% RSLogix 500 project JBT BIN SETTON ORIGINAL - COPY_BAK001.RSS, saved by version 10.00.00.00 %
PROJECT "JBT BIN"    % processor: MicroLogix 1200 %

PROGRAM FILES
  LAD 2   10 rungs
  LAD 3   7 rungs
  LAD 4   11 rungs
  LAD 5   33 rungs
  LAD 6   26 rungs
  LAD 7   16 rungs
  LAD 8   14 rungs
  LAD 9   43 rungs
  LAD 10   16 rungs
  LAD 11   9 rungs

DATA FILES
  O0 OUTPUT  6 elements
  I1 INPUT  6 elements
  S2 STATUS  66 elements
  B3 BINARY  5 elements
  T4 TIMER  35 elements
  C5 COUNTER  1 elements
  R6 CONTROL  1 elements
  N7 INTEGER  34 elements
  F8 FLOAT  1 elements
  L9   1 elements
  L10   2 elements

LADDER 2
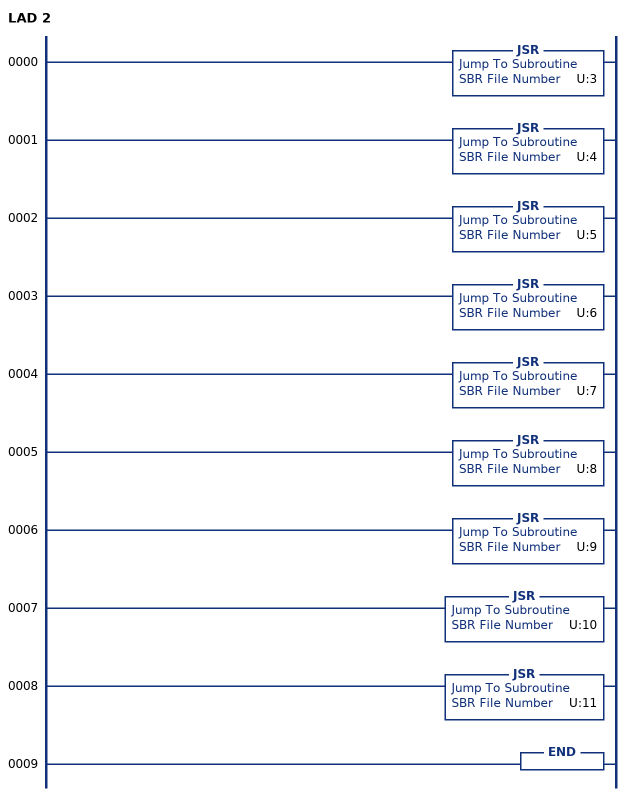
% Rung: 0 %
SOR JSR U:3 EOR
% Rung: 1 %
SOR JSR U:4 EOR
% Rung: 2 %
SOR JSR U:5 EOR
% Rung: 3 %
SOR JSR U:6 EOR
% Rung: 4 %
SOR JSR U:7 EOR
% Rung: 5 %
SOR JSR U:8 EOR
% Rung: 6 %
SOR JSR U:9 EOR
% Rung: 7 %
SOR JSR U:10 EOR
% Rung: 8 %
SOR JSR U:11 EOR
% Rung: 9 %
SOR END EOR

LADDER 3
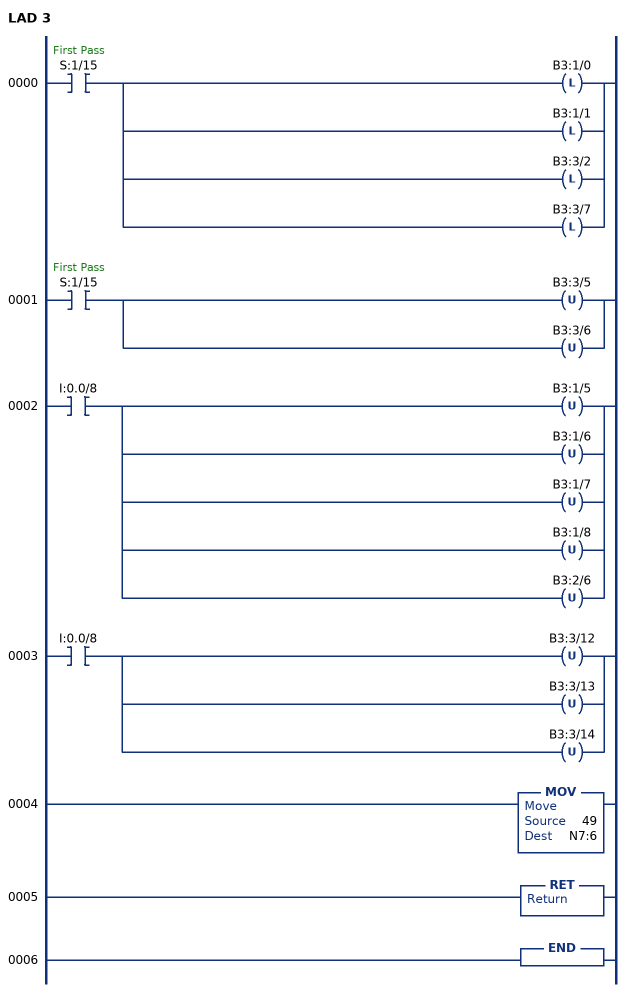
% Rung: 0 %
SOR XIC S:1/15 BST OTL B3:1/0 NXB BST OTL B3:1/1 NXB BST OTL B3:3/2 NXB OTL B3:3/7 BND BND BND EOR
%   S:1/15  "First Pass" %
% Rung: 1 %
SOR XIC S:1/15 BST OTU B3:3/5 NXB OTU B3:3/6 BND EOR
%   S:1/15  "First Pass" %
% Rung: 2 %
SOR XIC I:0.0/8 BST OTU B3:1/5 NXB BST OTU B3:1/6 NXB OTU B3:1/7 NXB BST OTU B3:1/8 NXB OTU B3:2/6 BND BND BND EOR
% Rung: 3 %
SOR XIC I:0.0/8 BST OTU B3:3/12 NXB OTU B3:3/13 NXB OTU B3:3/14 BND EOR
% Rung: 4 %
SOR MOV 49 N7:6 EOR
% Rung: 5 %
SOR RET EOR
% Rung: 6 %
SOR END EOR

LADDER 4
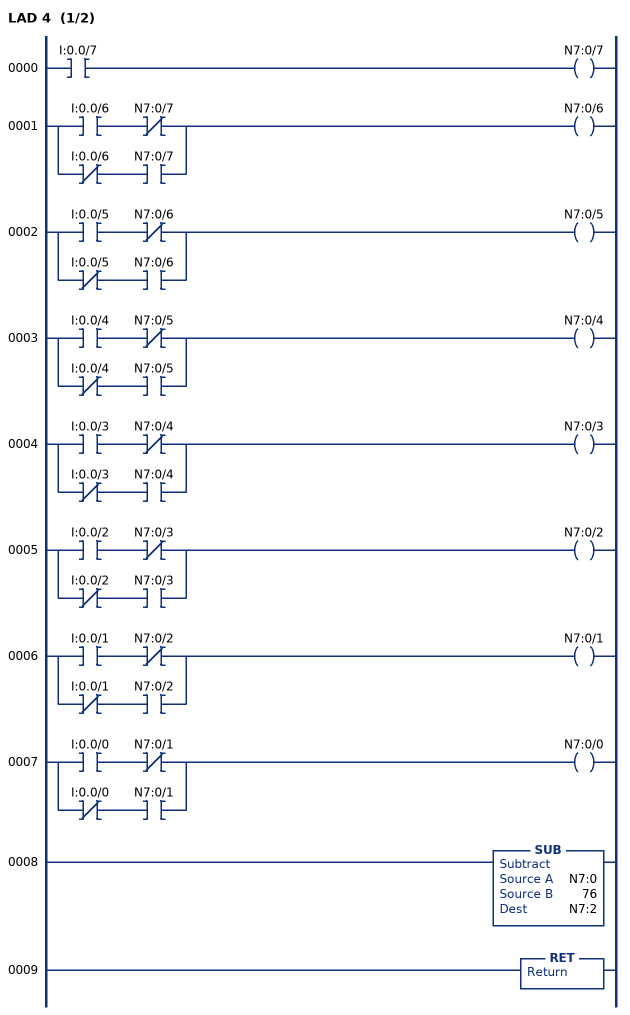
% Rung: 0 %
SOR XIC I:0.0/7 OTE N7:0/7 EOR
% Rung: 1 %
SOR BST XIC I:0.0/6 XIO N7:0/7 NXB XIO I:0.0/6 XIC N7:0/7 BND OTE N7:0/6 EOR
% Rung: 2 %
SOR BST XIC I:0.0/5 XIO N7:0/6 NXB XIO I:0.0/5 XIC N7:0/6 BND OTE N7:0/5 EOR
% Rung: 3 %
SOR BST XIC I:0.0/4 XIO N7:0/5 NXB XIO I:0.0/4 XIC N7:0/5 BND OTE N7:0/4 EOR
% Rung: 4 %
SOR BST XIC I:0.0/3 XIO N7:0/4 NXB XIO I:0.0/3 XIC N7:0/4 BND OTE N7:0/3 EOR
% Rung: 5 %
SOR BST XIC I:0.0/2 XIO N7:0/3 NXB XIO I:0.0/2 XIC N7:0/3 BND OTE N7:0/2 EOR
% Rung: 6 %
SOR BST XIC I:0.0/1 XIO N7:0/2 NXB XIO I:0.0/1 XIC N7:0/2 BND OTE N7:0/1 EOR
% Rung: 7 %
SOR BST XIC I:0.0/0 XIO N7:0/1 NXB XIO I:0.0/0 XIC N7:0/1 BND OTE N7:0/0 EOR
% Rung: 8 %
SOR SUB N7:0 76 N7:2 EOR
% Rung: 9 %
SOR RET EOR

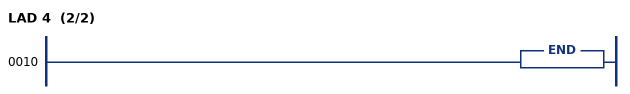
% Rung: 10 %
SOR END EOR

LADDER 5
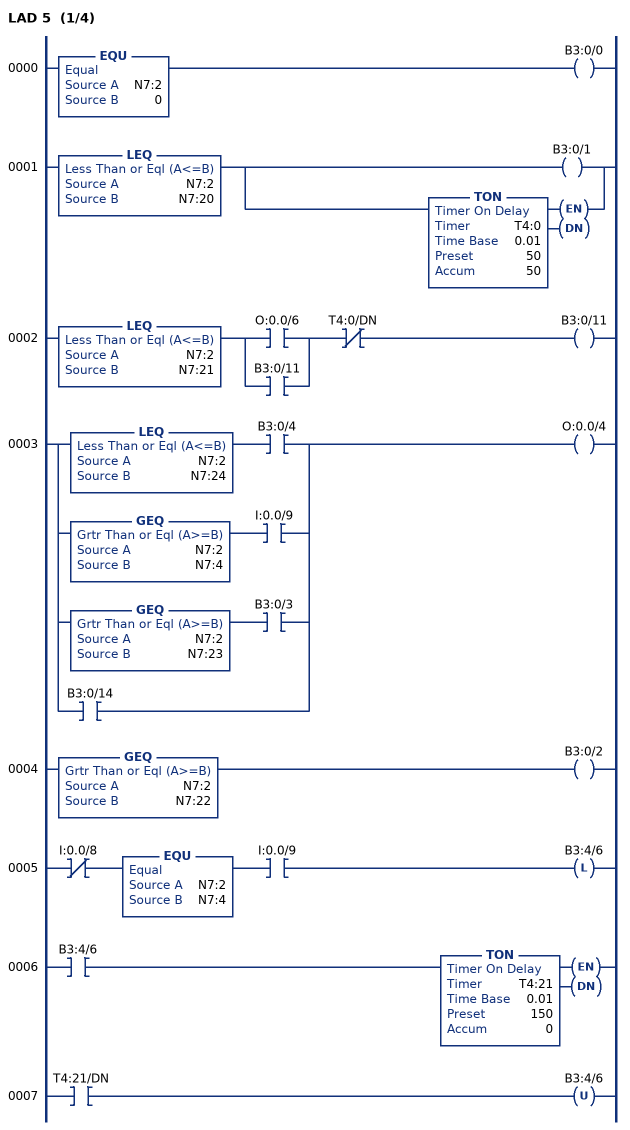
% Rung: 0 %
SOR EQU N7:2 0 OTE B3:0/0 EOR
% Rung: 1 %
SOR LEQ N7:2 N7:20 BST OTE B3:0/1 NXB TON T4:0 0.01 50 50 BND EOR
% Rung: 2 %
SOR LEQ N7:2 N7:21 BST XIC O:0.0/6 NXB XIC B3:0/11 BND XIO T4:0/DN OTE B3:0/11 EOR
% Rung: 3 %
SOR BST LEQ N7:2 N7:24 XIC B3:0/4 NXB GEQ N7:2 N7:4 XIC I:0.0/9 NXB BST GEQ N7:2 N7:23 XIC B3:0/3 NXB XIC B3:0/14 BND BND OTE O:0.0/4 EOR
% Rung: 4 %
SOR GEQ N7:2 N7:22 OTE B3:0/2 EOR
% Rung: 5 %
SOR XIO I:0.0/8 EQU N7:2 N7:4 XIC I:0.0/9 OTL B3:4/6 EOR
% Rung: 6 %
SOR XIC B3:4/6 TON T4:21 0.01 150 0 EOR
% Rung: 7 %
SOR XIC T4:21/DN OTU B3:4/6 EOR

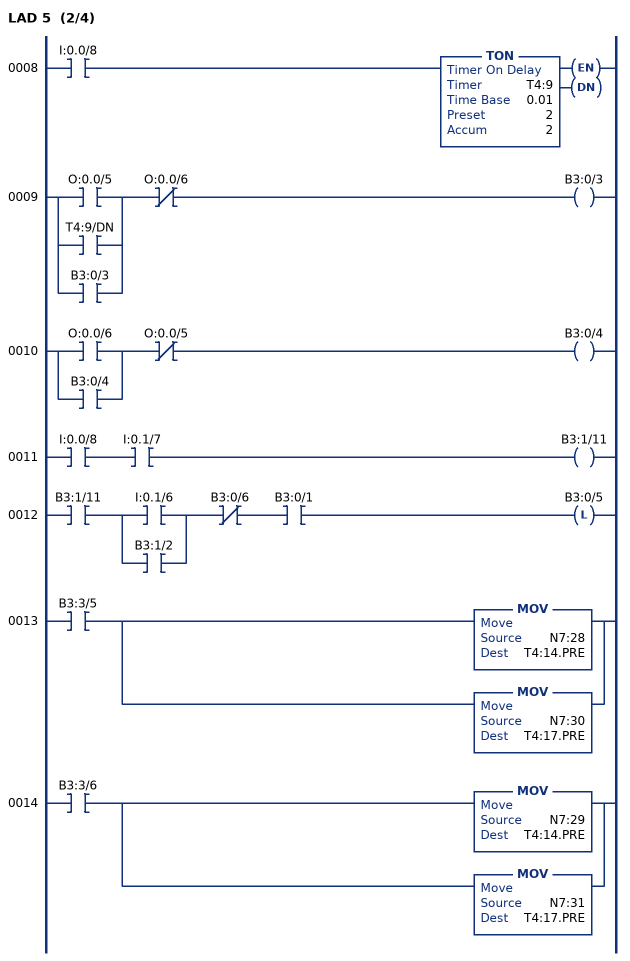
% Rung: 8 %
SOR XIC I:0.0/8 TON T4:9 0.01 2 2 EOR
% Rung: 9 %
SOR BST XIC O:0.0/5 NXB XIC T4:9/DN NXB XIC B3:0/3 BND XIO O:0.0/6 OTE B3:0/3 EOR
% Rung: 10 %
SOR BST XIC O:0.0/6 NXB XIC B3:0/4 BND XIO O:0.0/5 OTE B3:0/4 EOR
% Rung: 11 %
SOR XIC I:0.0/8 XIC I:0.1/7 OTE B3:1/11 EOR
% Rung: 12 %
SOR XIC B3:1/11 BST XIC I:0.1/6 NXB XIC B3:1/2 BND XIO B3:0/6 XIC B3:0/1 OTL B3:0/5 EOR
% Rung: 13 %
SOR XIC B3:3/5 BST MOV N7:28 T4:14.PRE NXB MOV N7:30 T4:17.PRE BND EOR
% Rung: 14 %
SOR XIC B3:3/6 BST MOV N7:29 T4:14.PRE NXB MOV N7:31 T4:17.PRE BND EOR

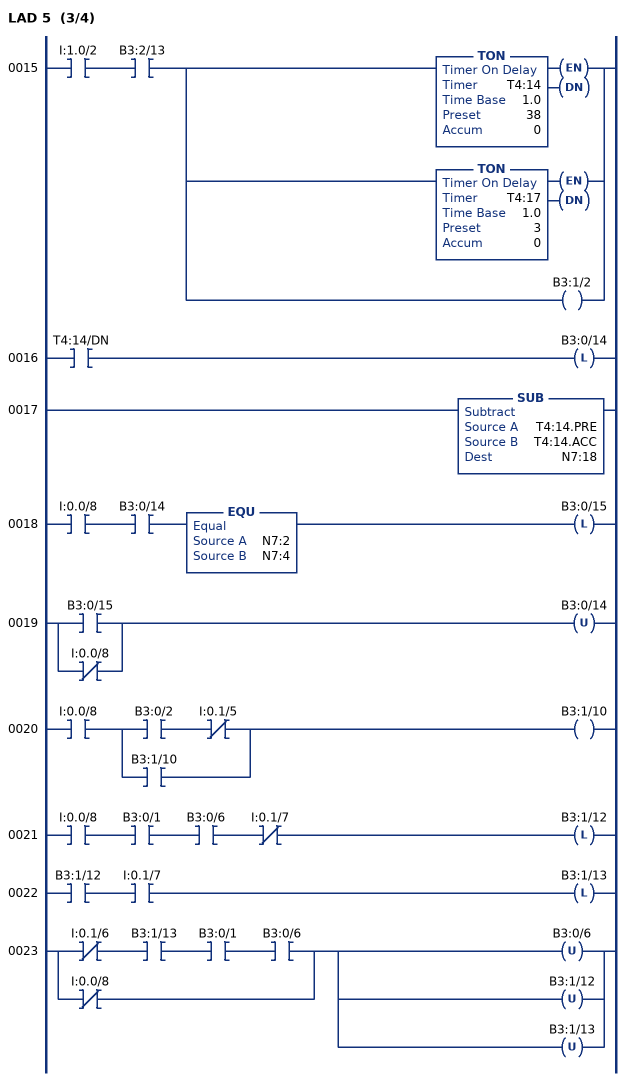
% Rung: 15 %
SOR XIC I:1.0/2 XIC B3:2/13 BST TON T4:14 1.0 38 0 NXB TON T4:17 1.0 3 0 NXB OTE B3:1/2 BND EOR
% Rung: 16 %
SOR XIC T4:14/DN OTL B3:0/14 EOR
% Rung: 17 %
SOR SUB T4:14.PRE T4:14.ACC N7:18 EOR
% Rung: 18 %
SOR XIC I:0.0/8 XIC B3:0/14 EQU N7:2 N7:4 OTL B3:0/15 EOR
% Rung: 19 %
SOR BST XIC B3:0/15 NXB XIO I:0.0/8 BND OTU B3:0/14 EOR
% Rung: 20 %
SOR XIC I:0.0/8 BST XIC B3:0/2 XIO I:0.1/5 NXB XIC B3:1/10 BND OTE B3:1/10 EOR
% Rung: 21 %
SOR XIC I:0.0/8 XIC B3:0/1 XIC B3:0/6 XIO I:0.1/7 OTL B3:1/12 EOR
% Rung: 22 %
SOR XIC B3:1/12 XIC I:0.1/7 OTL B3:1/13 EOR
% Rung: 23 %
SOR BST XIO I:0.1/6 XIC B3:1/13 XIC B3:0/1 XIC B3:0/6 NXB XIO I:0.0/8 BND BST OTU B3:0/6 NXB BST OTU B3:1/12 NXB OTU B3:1/13 BND BND EOR

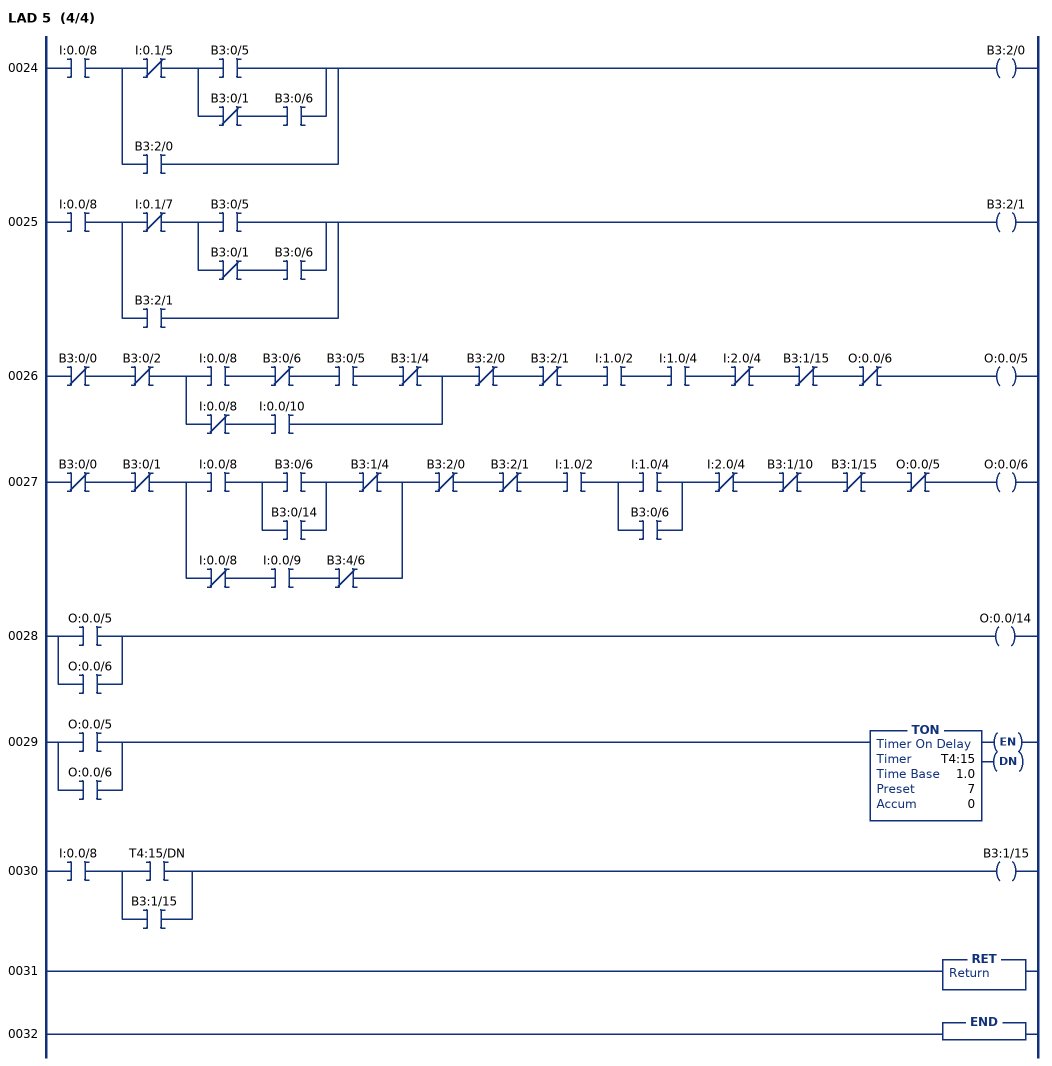
% Rung: 24 %
SOR XIC I:0.0/8 BST XIO I:0.1/5 BST XIC B3:0/5 NXB XIO B3:0/1 XIC B3:0/6 BND NXB XIC B3:2/0 BND OTE B3:2/0 EOR
% Rung: 25 %
SOR XIC I:0.0/8 BST XIO I:0.1/7 BST XIC B3:0/5 NXB XIO B3:0/1 XIC B3:0/6 BND NXB XIC B3:2/1 BND OTE B3:2/1 EOR
% Rung: 26 %
SOR XIO B3:0/0 XIO B3:0/2 BST XIC I:0.0/8 XIO B3:0/6 XIC B3:0/5 XIO B3:1/4 NXB XIO I:0.0/8 XIC I:0.0/10 BND XIO B3:2/0 XIO B3:2/1 XIC I:1.0/2 XIC I:1.0/4 XIO I:2.0/4 XIO B3:1/15 XIO O:0.0/6 OTE O:0.0/5 EOR
% Rung: 27 %
SOR XIO B3:0/0 XIO B3:0/1 BST XIC I:0.0/8 BST XIC B3:0/6 NXB XIC B3:0/14 BND XIO B3:1/4 NXB XIO I:0.0/8 XIC I:0.0/9 XIO B3:4/6 BND XIO B3:2/0 XIO B3:2/1 XIC I:1.0/2 BST XIC I:1.0/4 NXB XIC B3:0/6 BND XIO I:2.0/4 XIO B3:1/10 XIO B3:1/15 XIO O:0.0/5 OTE O:0.0/6 EOR
% Rung: 28 %
SOR BST XIC O:0.0/5 NXB XIC O:0.0/6 BND OTE O:0.0/14 EOR
% Rung: 29 %
SOR BST XIC O:0.0/5 NXB XIC O:0.0/6 BND TON T4:15 1.0 7 0 EOR
% Rung: 30 %
SOR XIC I:0.0/8 BST XIC T4:15/DN NXB XIC B3:1/15 BND OTE B3:1/15 EOR
% Rung: 31 %
SOR RET EOR
% Rung: 32 %
SOR END EOR

LADDER 6
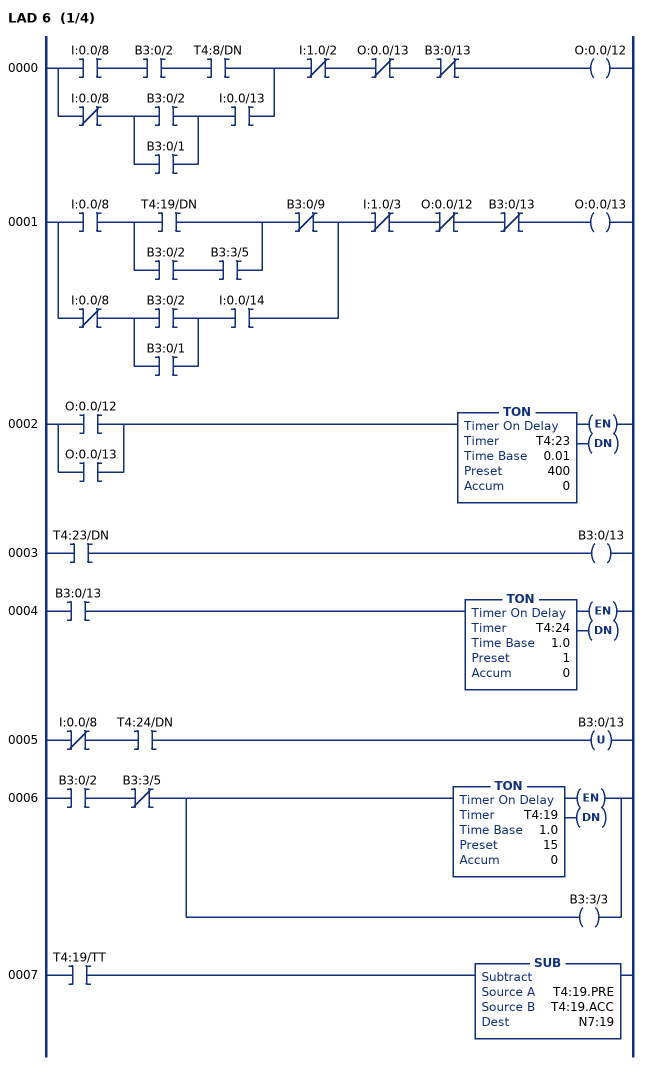
% Rung: 0 %
SOR BST XIC I:0.0/8 XIC B3:0/2 XIC T4:8/DN NXB XIO I:0.0/8 BST XIC B3:0/2 NXB XIC B3:0/1 BND XIC I:0.0/13 BND XIO I:1.0/2 XIO O:0.0/13 XIO B3:0/13 OTE O:0.0/12 EOR
% Rung: 1 %
SOR BST XIC I:0.0/8 BST XIC T4:19/DN NXB XIC B3:0/2 XIC B3:3/5 BND XIO B3:0/9 NXB XIO I:0.0/8 BST XIC B3:0/2 NXB XIC B3:0/1 BND XIC I:0.0/14 BND XIO I:1.0/3 XIO O:0.0/12 XIO B3:0/13 OTE O:0.0/13 EOR
% Rung: 2 %
SOR BST XIC O:0.0/12 NXB XIC O:0.0/13 BND TON T4:23 0.01 400 0 EOR
% Rung: 3 %
SOR XIC T4:23/DN OTE B3:0/13 EOR
% Rung: 4 %
SOR XIC B3:0/13 TON T4:24 1.0 1 0 EOR
% Rung: 5 %
SOR XIO I:0.0/8 XIC T4:24/DN OTU B3:0/13 EOR
% Rung: 6 %
SOR XIC B3:0/2 XIO B3:3/5 BST TON T4:19 1.0 15 0 NXB OTE B3:3/3 BND EOR
% Rung: 7 %
SOR XIC T4:19/TT SUB T4:19.PRE T4:19.ACC N7:19 EOR

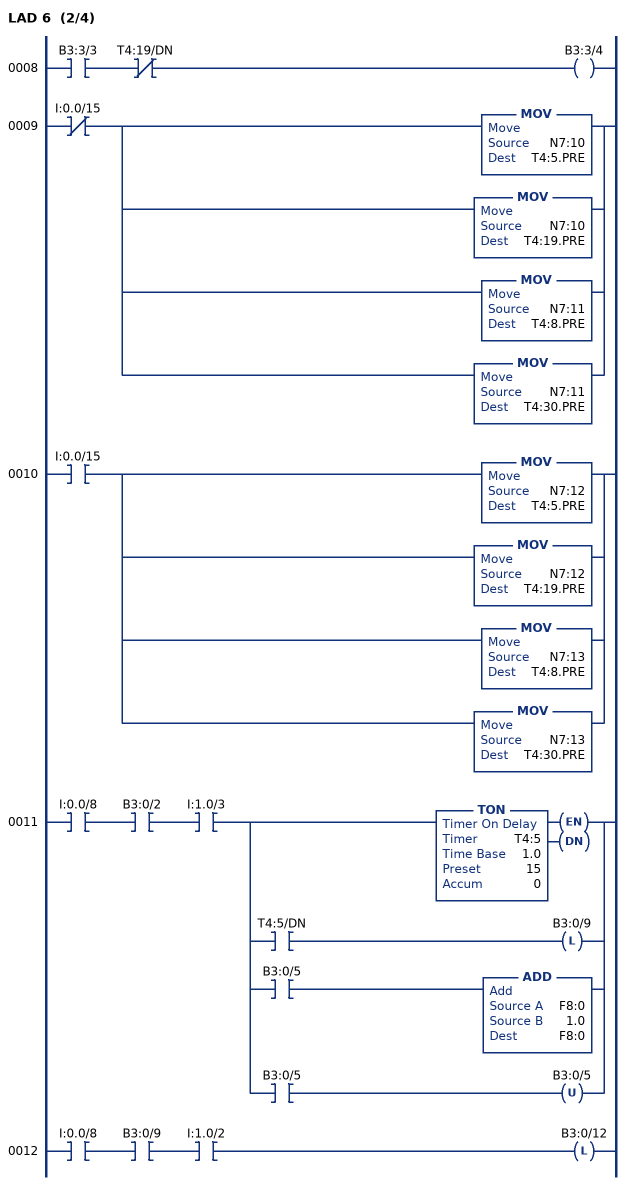
% Rung: 8 %
SOR XIC B3:3/3 XIO T4:19/DN OTE B3:3/4 EOR
% Rung: 9 %
SOR XIO I:0.0/15 BST MOV N7:10 T4:5.PRE NXB MOV N7:10 T4:19.PRE NXB MOV N7:11 T4:8.PRE NXB MOV N7:11 T4:30.PRE BND EOR
% Rung: 10 %
SOR XIC I:0.0/15 BST MOV N7:12 T4:5.PRE NXB MOV N7:12 T4:19.PRE NXB MOV N7:13 T4:8.PRE NXB MOV N7:13 T4:30.PRE BND EOR
% Rung: 11 %
SOR XIC I:0.0/8 XIC B3:0/2 XIC I:1.0/3 BST TON T4:5 1.0 15 0 NXB XIC T4:5/DN OTL B3:0/9 NXB BST XIC B3:0/5 ADD F8:0 1.0 F8:0 NXB XIC B3:0/5 OTU B3:0/5 BND BND EOR
% Rung: 12 %
SOR XIC I:0.0/8 XIC B3:0/9 XIC I:1.0/2 OTL B3:0/12 EOR

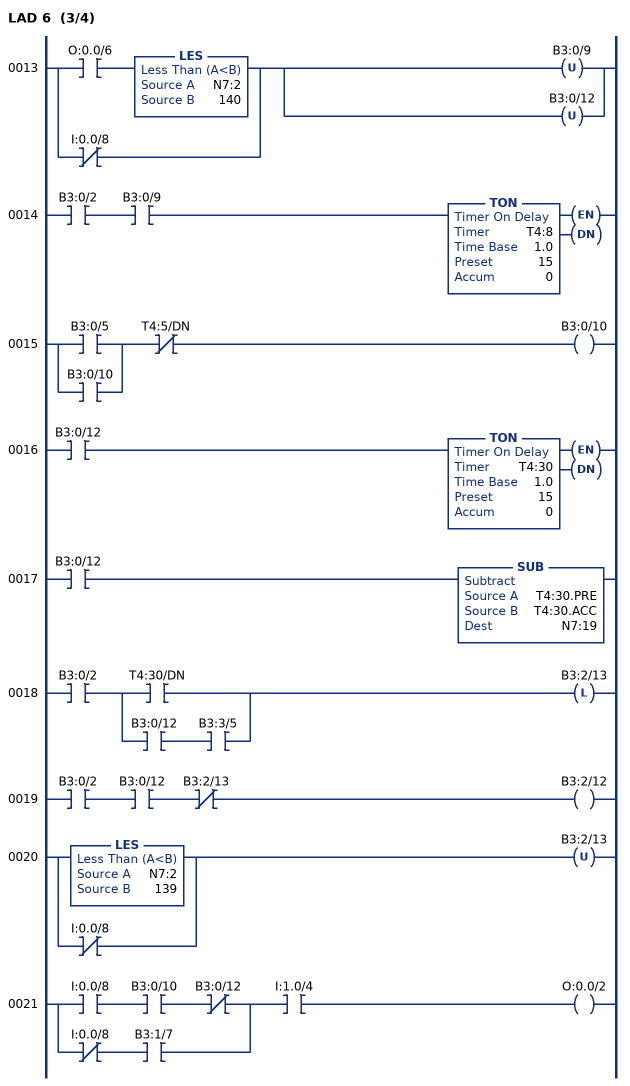
% Rung: 13 %
SOR BST XIC O:0.0/6 LES N7:2 140 NXB XIO I:0.0/8 BND BST OTU B3:0/9 NXB OTU B3:0/12 BND EOR
% Rung: 14 %
SOR XIC B3:0/2 XIC B3:0/9 TON T4:8 1.0 15 0 EOR
% Rung: 15 %
SOR BST XIC B3:0/5 NXB XIC B3:0/10 BND XIO T4:5/DN OTE B3:0/10 EOR
% Rung: 16 %
SOR XIC B3:0/12 TON T4:30 1.0 15 0 EOR
% Rung: 17 %
SOR XIC B3:0/12 SUB T4:30.PRE T4:30.ACC N7:19 EOR
% Rung: 18 %
SOR XIC B3:0/2 BST XIC T4:30/DN NXB XIC B3:0/12 XIC B3:3/5 BND OTL B3:2/13 EOR
% Rung: 19 %
SOR XIC B3:0/2 XIC B3:0/12 XIO B3:2/13 OTE B3:2/12 EOR
% Rung: 20 %
SOR BST LES N7:2 139 NXB XIO I:0.0/8 BND OTU B3:2/13 EOR
% Rung: 21 %
SOR BST XIC I:0.0/8 XIC B3:0/10 XIO B3:0/12 NXB XIO I:0.0/8 XIC B3:1/7 BND XIC I:1.0/4 OTE O:0.0/2 EOR

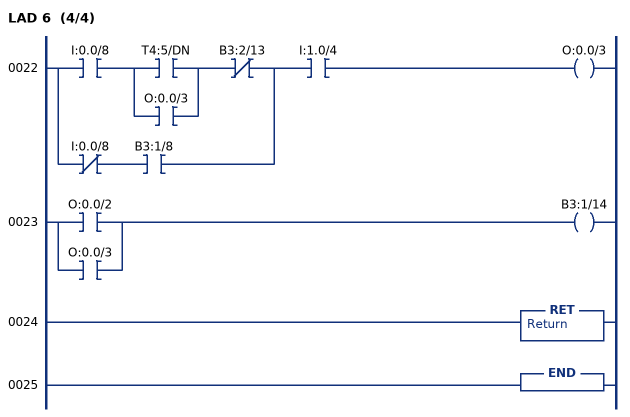
% Rung: 22 %
SOR BST XIC I:0.0/8 BST XIC T4:5/DN NXB XIC O:0.0/3 BND XIO B3:2/13 NXB XIO I:0.0/8 XIC B3:1/8 BND XIC I:1.0/4 OTE O:0.0/3 EOR
% Rung: 23 %
SOR BST XIC O:0.0/2 NXB XIC O:0.0/3 BND OTE B3:1/14 EOR
% Rung: 24 %
SOR RET EOR
% Rung: 25 %
SOR END EOR

LADDER 7
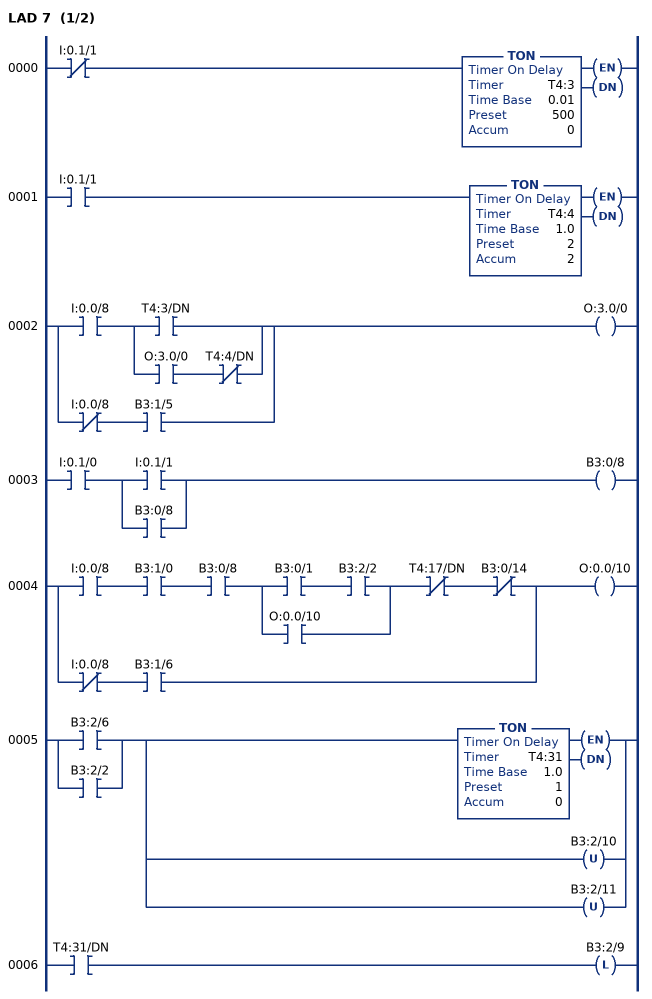
% Rung: 0 %
SOR XIO I:0.1/1 TON T4:3 0.01 500 0 EOR
% Rung: 1 %
SOR XIC I:0.1/1 TON T4:4 1.0 2 2 EOR
% Rung: 2 %
SOR BST XIC I:0.0/8 BST XIC T4:3/DN NXB XIC O:3.0/0 XIO T4:4/DN BND NXB XIO I:0.0/8 XIC B3:1/5 BND OTE O:3.0/0 EOR
% Rung: 3 %
SOR XIC I:0.1/0 BST XIC I:0.1/1 NXB XIC B3:0/8 BND OTE B3:0/8 EOR
% Rung: 4 %
SOR BST XIC I:0.0/8 XIC B3:1/0 XIC B3:0/8 BST XIC B3:0/1 XIC B3:2/2 NXB XIC O:0.0/10 BND XIO T4:17/DN XIO B3:0/14 NXB XIO I:0.0/8 XIC B3:1/6 BND OTE O:0.0/10 EOR
% Rung: 5 %
SOR BST XIC B3:2/6 NXB XIC B3:2/2 BND BST TON T4:31 1.0 1 0 NXB BST OTU B3:2/10 NXB OTU B3:2/11 BND BND EOR
% Rung: 6 %
SOR XIC T4:31/DN OTL B3:2/9 EOR

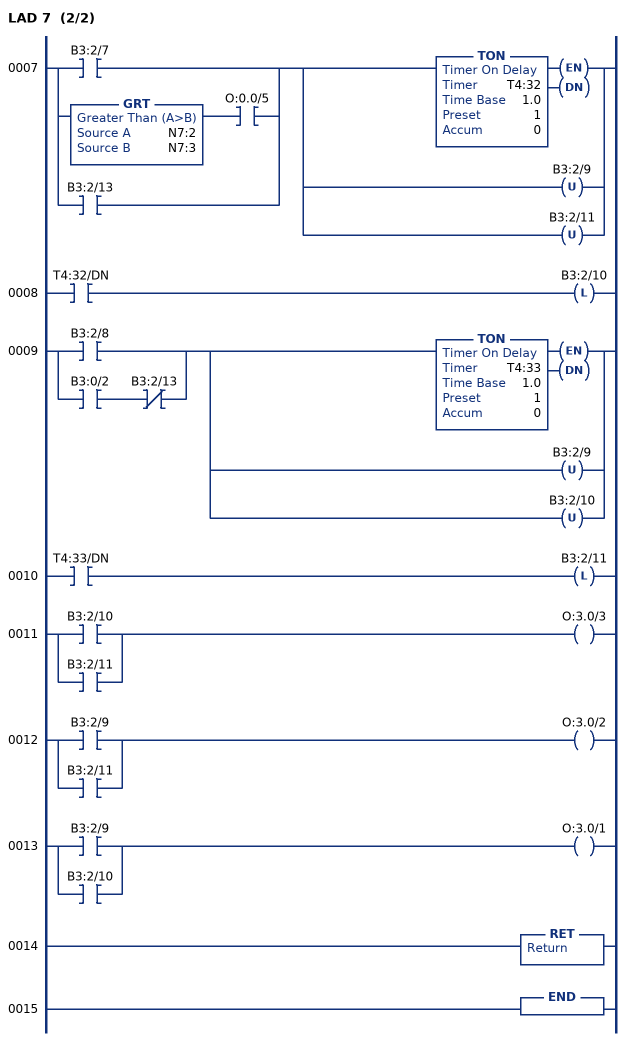
% Rung: 7 %
SOR BST BST XIC B3:2/7 NXB GRT N7:2 N7:3 XIC O:0.0/5 BND NXB XIC B3:2/13 BND BST TON T4:32 1.0 1 0 NXB BST OTU B3:2/9 NXB OTU B3:2/11 BND BND EOR
% Rung: 8 %
SOR XIC T4:32/DN OTL B3:2/10 EOR
% Rung: 9 %
SOR BST XIC B3:2/8 NXB XIC B3:0/2 XIO B3:2/13 BND BST TON T4:33 1.0 1 0 NXB BST OTU B3:2/9 NXB OTU B3:2/10 BND BND EOR
% Rung: 10 %
SOR XIC T4:33/DN OTL B3:2/11 EOR
% Rung: 11 %
SOR BST XIC B3:2/10 NXB XIC B3:2/11 BND OTE O:3.0/3 EOR
% Rung: 12 %
SOR BST XIC B3:2/9 NXB XIC B3:2/11 BND OTE O:3.0/2 EOR
% Rung: 13 %
SOR BST XIC B3:2/9 NXB XIC B3:2/10 BND OTE O:3.0/1 EOR
% Rung: 14 %
SOR RET EOR
% Rung: 15 %
SOR END EOR

LADDER 8
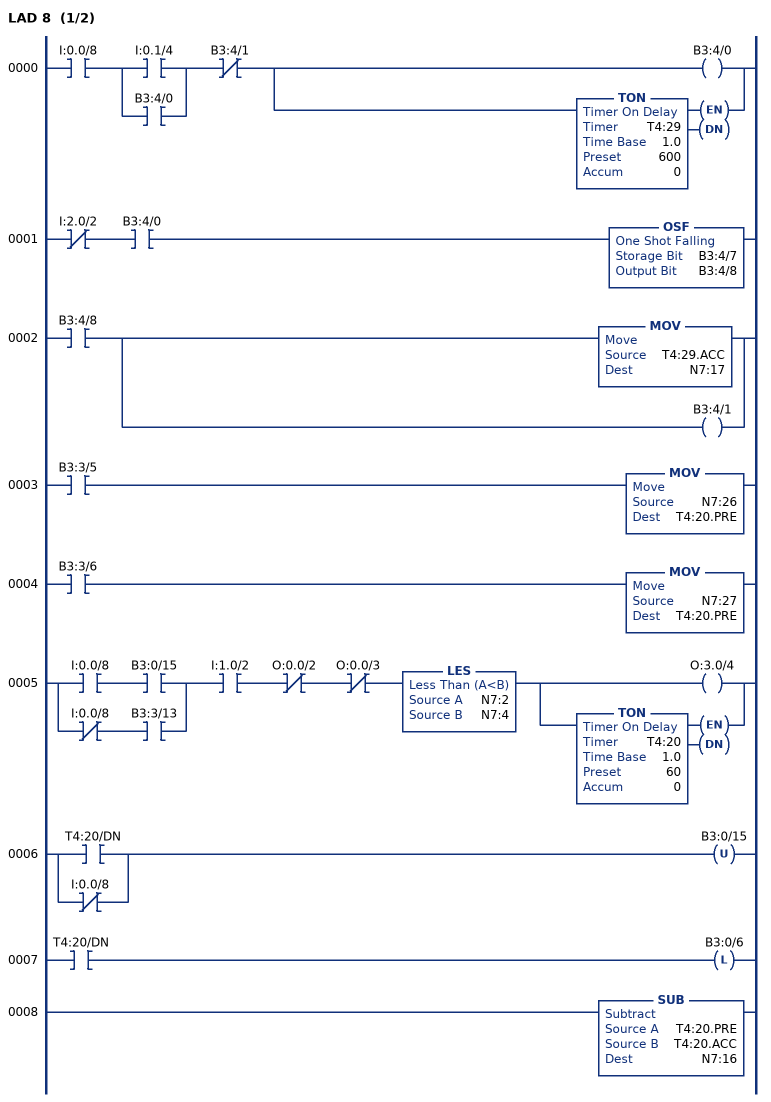
% Rung: 0 %
SOR XIC I:0.0/8 BST XIC I:0.1/4 NXB XIC B3:4/0 BND XIO B3:4/1 BST OTE B3:4/0 NXB TON T4:29 1.0 600 0 BND EOR
% Rung: 1 %
SOR XIO I:2.0/2 XIC B3:4/0 OSF B3:4/7 B3:4/8 EOR
% Rung: 2 %
SOR XIC B3:4/8 BST MOV T4:29.ACC N7:17 NXB OTE B3:4/1 BND EOR
% Rung: 3 %
SOR XIC B3:3/5 MOV N7:26 T4:20.PRE EOR
% Rung: 4 %
SOR XIC B3:3/6 MOV N7:27 T4:20.PRE EOR
% Rung: 5 %
SOR BST XIC I:0.0/8 XIC B3:0/15 NXB XIO I:0.0/8 XIC B3:3/13 BND XIC I:1.0/2 XIO O:0.0/2 XIO O:0.0/3 LES N7:2 N7:4 BST OTE O:3.0/4 NXB TON T4:20 1.0 60 0 BND EOR
% Rung: 6 %
SOR BST XIC T4:20/DN NXB XIO I:0.0/8 BND OTU B3:0/15 EOR
% Rung: 7 %
SOR XIC T4:20/DN OTL B3:0/6 EOR
% Rung: 8 %
SOR SUB T4:20.PRE T4:20.ACC N7:16 EOR

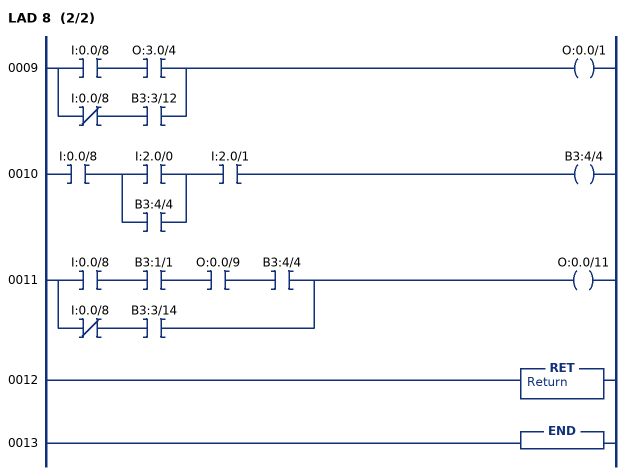
% Rung: 9 %
SOR BST XIC I:0.0/8 XIC O:3.0/4 NXB XIO I:0.0/8 XIC B3:3/12 BND OTE O:0.0/1 EOR
% Rung: 10 %
SOR XIC I:0.0/8 BST XIC I:2.0/0 NXB XIC B3:4/4 BND XIC I:2.0/1 OTE B3:4/4 EOR
% Rung: 11 %
SOR BST XIC I:0.0/8 XIC B3:1/1 XIC O:0.0/9 XIC B3:4/4 NXB XIO I:0.0/8 XIC B3:3/14 BND OTE O:0.0/11 EOR
% Rung: 12 %
SOR RET EOR
% Rung: 13 %
SOR END EOR

LADDER 9
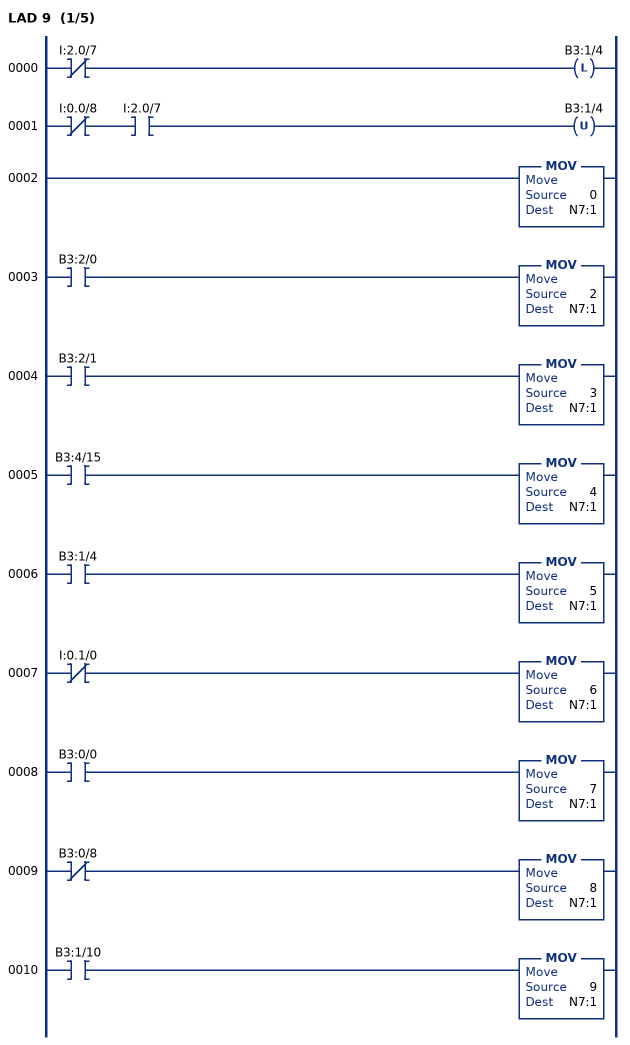
% Rung: 0 %
SOR XIO I:2.0/7 OTL B3:1/4 EOR
% Rung: 1 %
SOR XIO I:0.0/8 XIC I:2.0/7 OTU B3:1/4 EOR
% Rung: 2 %
SOR MOV 0 N7:1 EOR
% Rung: 3 %
SOR XIC B3:2/0 MOV 2 N7:1 EOR
% Rung: 4 %
SOR XIC B3:2/1 MOV 3 N7:1 EOR
% Rung: 5 %
SOR XIC B3:4/15 MOV 4 N7:1 EOR
% Rung: 6 %
SOR XIC B3:1/4 MOV 5 N7:1 EOR
% Rung: 7 %
SOR XIO I:0.1/0 MOV 6 N7:1 EOR
% Rung: 8 %
SOR XIC B3:0/0 MOV 7 N7:1 EOR
% Rung: 9 %
SOR XIO B3:0/8 MOV 8 N7:1 EOR
% Rung: 10 %
SOR XIC B3:1/10 MOV 9 N7:1 EOR

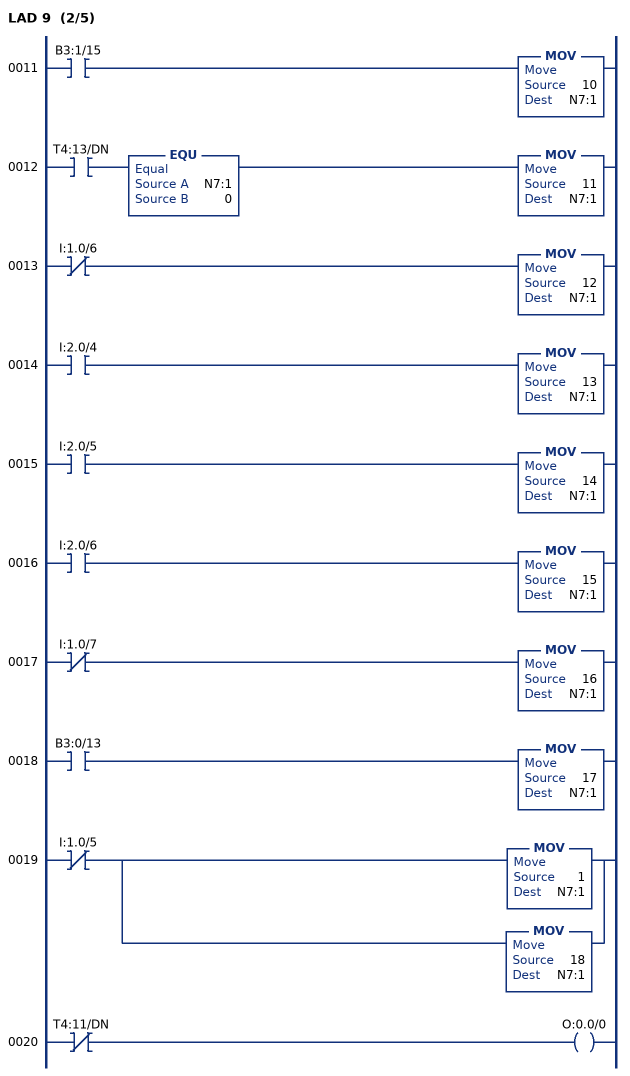
% Rung: 11 %
SOR XIC B3:1/15 MOV 10 N7:1 EOR
% Rung: 12 %
SOR XIC T4:13/DN EQU N7:1 0 MOV 11 N7:1 EOR
% Rung: 13 %
SOR XIO I:1.0/6 MOV 12 N7:1 EOR
% Rung: 14 %
SOR XIC I:2.0/4 MOV 13 N7:1 EOR
% Rung: 15 %
SOR XIC I:2.0/5 MOV 14 N7:1 EOR
% Rung: 16 %
SOR XIC I:2.0/6 MOV 15 N7:1 EOR
% Rung: 17 %
SOR XIO I:1.0/7 MOV 16 N7:1 EOR
% Rung: 18 %
SOR XIC B3:0/13 MOV 17 N7:1 EOR
% Rung: 19 %
SOR XIO I:1.0/5 BST MOV 1 N7:1 NXB MOV 18 N7:1 BND EOR
% Rung: 20 %
SOR XIO T4:11/DN OTE O:0.0/0 EOR

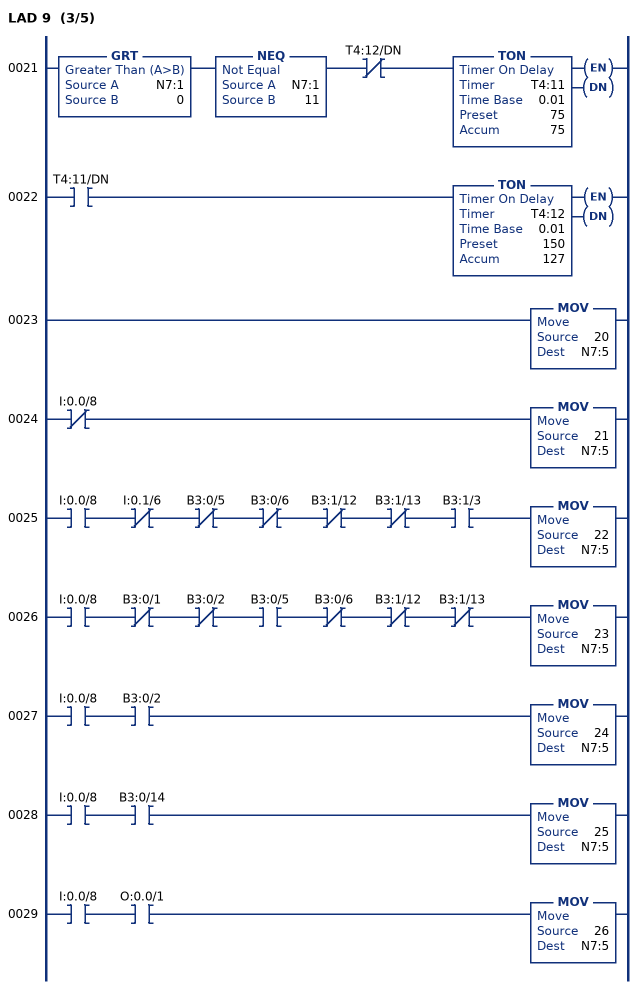
% Rung: 21 %
SOR GRT N7:1 0 NEQ N7:1 11 XIO T4:12/DN TON T4:11 0.01 75 75 EOR
% Rung: 22 %
SOR XIC T4:11/DN TON T4:12 0.01 150 127 EOR
% Rung: 23 %
SOR MOV 20 N7:5 EOR
% Rung: 24 %
SOR XIO I:0.0/8 MOV 21 N7:5 EOR
% Rung: 25 %
SOR XIC I:0.0/8 XIO I:0.1/6 XIO B3:0/5 XIO B3:0/6 XIO B3:1/12 XIO B3:1/13 XIC B3:1/3 MOV 22 N7:5 EOR
% Rung: 26 %
SOR XIC I:0.0/8 XIO B3:0/1 XIO B3:0/2 XIC B3:0/5 XIO B3:0/6 XIO B3:1/12 XIO B3:1/13 MOV 23 N7:5 EOR
% Rung: 27 %
SOR XIC I:0.0/8 XIC B3:0/2 MOV 24 N7:5 EOR
% Rung: 28 %
SOR XIC I:0.0/8 XIC B3:0/14 MOV 25 N7:5 EOR
% Rung: 29 %
SOR XIC I:0.0/8 XIC O:0.0/1 MOV 26 N7:5 EOR

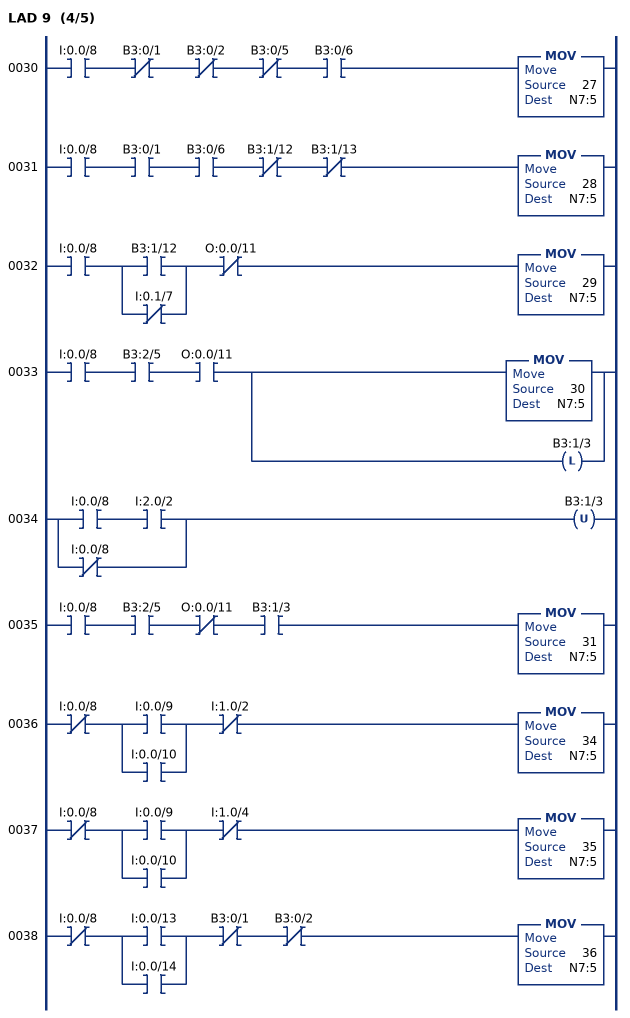
% Rung: 30 %
SOR XIC I:0.0/8 XIO B3:0/1 XIO B3:0/2 XIO B3:0/5 XIC B3:0/6 MOV 27 N7:5 EOR
% Rung: 31 %
SOR XIC I:0.0/8 XIC B3:0/1 XIC B3:0/6 XIO B3:1/12 XIO B3:1/13 MOV 28 N7:5 EOR
% Rung: 32 %
SOR XIC I:0.0/8 BST XIC B3:1/12 NXB XIO I:0.1/7 BND XIO O:0.0/11 MOV 29 N7:5 EOR
% Rung: 33 %
SOR XIC I:0.0/8 XIC B3:2/5 XIC O:0.0/11 BST MOV 30 N7:5 NXB OTL B3:1/3 BND EOR
% Rung: 34 %
SOR BST XIC I:0.0/8 XIC I:2.0/2 NXB XIO I:0.0/8 BND OTU B3:1/3 EOR
% Rung: 35 %
SOR XIC I:0.0/8 XIC B3:2/5 XIO O:0.0/11 XIC B3:1/3 MOV 31 N7:5 EOR
% Rung: 36 %
SOR XIO I:0.0/8 BST XIC I:0.0/9 NXB XIC I:0.0/10 BND XIO I:1.0/2 MOV 34 N7:5 EOR
% Rung: 37 %
SOR XIO I:0.0/8 BST XIC I:0.0/9 NXB XIC I:0.0/10 BND XIO I:1.0/4 MOV 35 N7:5 EOR
% Rung: 38 %
SOR XIO I:0.0/8 BST XIC I:0.0/13 NXB XIC I:0.0/14 BND XIO B3:0/1 XIO B3:0/2 MOV 36 N7:5 EOR

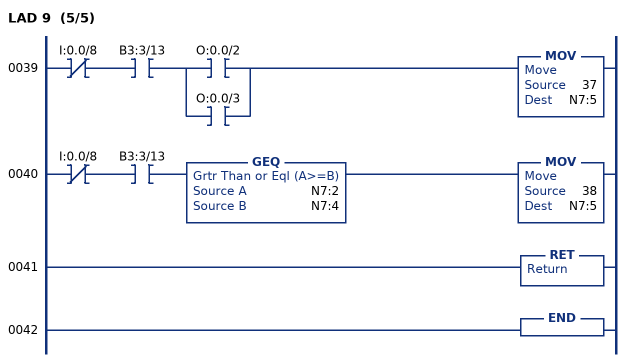
% Rung: 39 %
SOR XIO I:0.0/8 XIC B3:3/13 BST XIC O:0.0/2 NXB XIC O:0.0/3 BND MOV 37 N7:5 EOR
% Rung: 40 %
SOR XIO I:0.0/8 XIC B3:3/13 GEQ N7:2 N7:4 MOV 38 N7:5 EOR
% Rung: 41 %
SOR RET EOR
% Rung: 42 %
SOR END EOR

LADDER 10
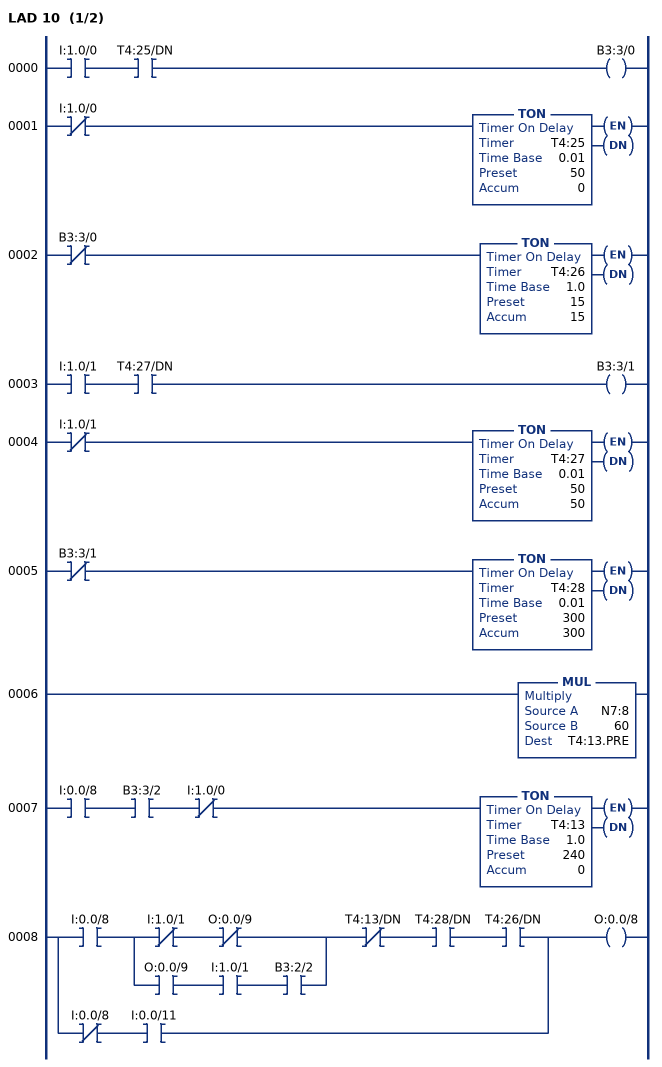
% Rung: 0 %
SOR XIC I:1.0/0 XIC T4:25/DN OTE B3:3/0 EOR
% Rung: 1 %
SOR XIO I:1.0/0 TON T4:25 0.01 50 0 EOR
% Rung: 2 %
SOR XIO B3:3/0 TON T4:26 1.0 15 15 EOR
% Rung: 3 %
SOR XIC I:1.0/1 XIC T4:27/DN OTE B3:3/1 EOR
% Rung: 4 %
SOR XIO I:1.0/1 TON T4:27 0.01 50 50 EOR
% Rung: 5 %
SOR XIO B3:3/1 TON T4:28 0.01 300 300 EOR
% Rung: 6 %
SOR MUL N7:8 60 T4:13.PRE EOR
% Rung: 7 %
SOR XIC I:0.0/8 XIC B3:3/2 XIO I:1.0/0 TON T4:13 1.0 240 0 EOR
% Rung: 8 %
SOR BST XIC I:0.0/8 BST XIO I:1.0/1 XIO O:0.0/9 NXB XIC O:0.0/9 XIC I:1.0/1 XIC B3:2/2 BND XIO T4:13/DN XIC T4:28/DN XIC T4:26/DN NXB XIO I:0.0/8 XIC I:0.0/11 BND OTE O:0.0/8 EOR

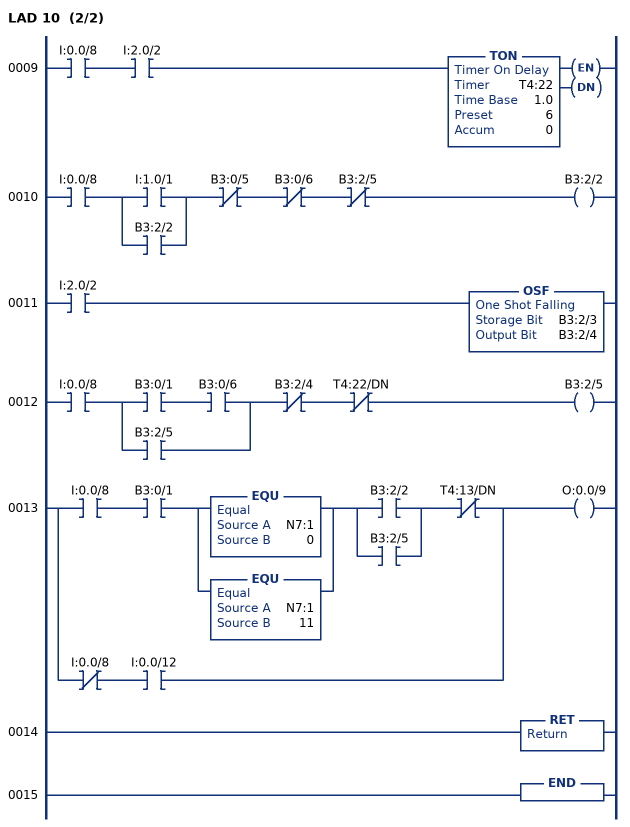
% Rung: 9 %
SOR XIC I:0.0/8 XIC I:2.0/2 TON T4:22 1.0 6 0 EOR
% Rung: 10 %
SOR XIC I:0.0/8 BST XIC I:1.0/1 NXB XIC B3:2/2 BND XIO B3:0/5 XIO B3:0/6 XIO B3:2/5 OTE B3:2/2 EOR
% Rung: 11 %
SOR XIC I:2.0/2 OSF B3:2/3 B3:2/4 EOR
% Rung: 12 %
SOR XIC I:0.0/8 BST XIC B3:0/1 XIC B3:0/6 NXB XIC B3:2/5 BND XIO B3:2/4 XIO T4:22/DN OTE B3:2/5 EOR
% Rung: 13 %
SOR BST XIC I:0.0/8 XIC B3:0/1 BST EQU N7:1 0 NXB EQU N7:1 11 BND BST XIC B3:2/2 NXB XIC B3:2/5 BND XIO T4:13/DN NXB XIO I:0.0/8 XIC I:0.0/12 BND OTE O:0.0/9 EOR
% Rung: 14 %
SOR RET EOR
% Rung: 15 %
SOR END EOR

LADDER 11
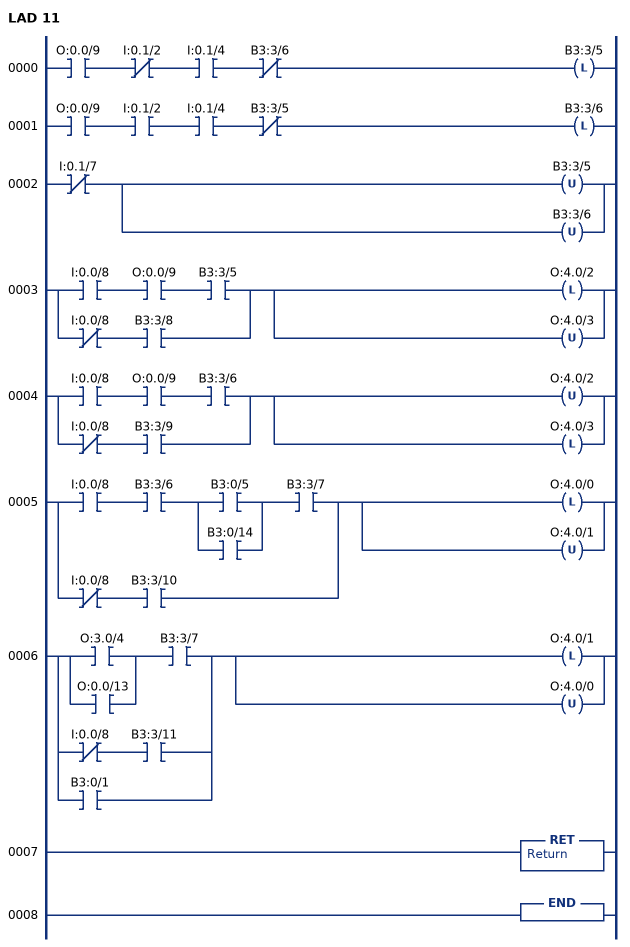
% Rung: 0 %
SOR XIC O:0.0/9 XIO I:0.1/2 XIC I:0.1/4 XIO B3:3/6 OTL B3:3/5 EOR
% Rung: 1 %
SOR XIC O:0.0/9 XIC I:0.1/2 XIC I:0.1/4 XIO B3:3/5 OTL B3:3/6 EOR
% Rung: 2 %
SOR XIO I:0.1/7 BST OTU B3:3/5 NXB OTU B3:3/6 BND EOR
% Rung: 3 %
SOR BST XIC I:0.0/8 XIC O:0.0/9 XIC B3:3/5 NXB XIO I:0.0/8 XIC B3:3/8 BND BST OTL O:4.0/2 NXB OTU O:4.0/3 BND EOR
% Rung: 4 %
SOR BST XIC I:0.0/8 XIC O:0.0/9 XIC B3:3/6 NXB XIO I:0.0/8 XIC B3:3/9 BND BST OTU O:4.0/2 NXB OTL O:4.0/3 BND EOR
% Rung: 5 %
SOR BST XIC I:0.0/8 XIC B3:3/6 BST XIC B3:0/5 NXB XIC B3:0/14 BND XIC B3:3/7 NXB XIO I:0.0/8 XIC B3:3/10 BND BST OTL O:4.0/0 NXB OTU O:4.0/1 BND EOR
% Rung: 6 %
SOR BST BST BST XIC O:3.0/4 NXB XIC O:0.0/13 BND XIC B3:3/7 NXB XIO I:0.0/8 XIC B3:3/11 BND NXB XIC B3:0/1 BND BST OTL O:4.0/1 NXB OTU O:4.0/0 BND EOR
% Rung: 7 %
SOR RET EOR
% Rung: 8 %
SOR END EOR

REVISION NOTES
  0: side pressure

DATA TABLE (non-zero values as saved)
DATA B3
% B3:0 % 0X011A 0X0803 0X0400 0X0084 0X0000
DATA T4
% .PRE .ACC %
% T4:0 % 50 50
% T4:1 % 1 0
% T4:2 % 1 0
% T4:3 % 500 0
% T4:4 % 2 2
% T4:5 % 15 0
% T4:6 % 658 0
% T4:7 % 375 500
% T4:8 % 15 0
% T4:9 % 2 2
% T4:10 % 500 0
% T4:11 % 75 75
% T4:12 % 150 127
% T4:13 % 240 0
% T4:14 % 38 0
% T4:15 % 7 0
% T4:16 % 6 0
% T4:17 % 3 0
% T4:18 % 100 0
% T4:19 % 15 0
% T4:20 % 60 0
% T4:21 % 150 0
% T4:22 % 6 0
% T4:23 % 400 0
% T4:24 % 1 0
% T4:25 % 50 0
% T4:26 % 15 15
% T4:27 % 50 50
% T4:28 % 300 300
% T4:29 % 600 0
% T4:30 % 15 0
% T4:31 % 1 0
% T4:32 % 1 0
% T4:33 % 1 0
DATA N7
% N7:0 % 85 18 9 20 106 20 49 0 4 0
% N7:10 % 8 7 15 15 0 0 60 190 38 0
% N7:20 % 10 12 141 105 45 0 60 60 38 38
% N7:30 % 3 3 0 0
DATA F8
% F8:0 % 363
